DATA_BLOCK "DigiforceMain_DB"   // DB47
VERSION : 0.1
// stored: AutoNumber true, DBAccessibleFromOPCUA true, DBAccessibleFromWebserver true, InstanceOfName DigiforceMain, InstanceOfType FB
"DigiforceMain"
BEGIN
   Digiforce1_Instance.DataRead := 488;
   Digiforce1_Instance.DataWrite := 487;
   Digiforce1_Instance.send.Tare_X := FALSE;
   Digiforce1_Instance.send.Res_Stat := FALSE;
   Digiforce1_Instance.send.Stest := FALSE;
   Digiforce1_Instance.send.Strobe := FALSE;
   Digiforce1_Instance.send.Auto := FALSE;
   Digiforce1_Instance.send.reserve1 := FALSE;
   Digiforce1_Instance.send.reserve2 := FALSE;
   Digiforce1_Instance.send.reserve3 := FALSE;
   Digiforce1_Instance.send.Prog := 16#00;
   Digiforce1_Instance.send.Start := FALSE;
   Digiforce1_Instance.receive.dataD.Ready := TRUE;
   Digiforce1_Instance.receive.dataD.OK := FALSE;
   Digiforce1_Instance.receive.dataD.NOK := TRUE;
   Digiforce1_Instance.receive.dataD.NOK_ONL := FALSE;
   Digiforce1_Instance.receive.dataD.S1 := TRUE;
   Digiforce1_Instance.receive.dataD.S2 := FALSE;
   Digiforce1_Instance.receive.dataD.OK_STEST := FALSE;
   Digiforce1_Instance.receive.dataD.MEAS_ACT := FALSE;
   Digiforce1_Instance.receive.dataD.Strobe := FALSE;
   Digiforce1_Instance.receive.dataD.Prog0 := FALSE;
   Digiforce1_Instance.receive.dataD.Prog1 := FALSE;
   Digiforce1_Instance.receive.dataD.Prog2 := FALSE;
   Digiforce1_Instance.receive.dataD.reserve1 := FALSE;
   Digiforce1_Instance.receive.dataD.reserve2 := FALSE;
   Digiforce1_Instance.receive.dataD.reserve3 := FALSE;
   Digiforce1_Instance.receive.dataD.reserve4 := FALSE;
   Digiforce1_Instance.receive.dataD.Global_NOK := TRUE;
   Digiforce1_Instance.receive.dataD."Overload _NOK" := FALSE;
   Digiforce1_Instance.receive.dataD.Window_1_NOK := TRUE;
   Digiforce1_Instance.receive.dataD.Window_2_NOK := FALSE;
   Digiforce1_Instance.receive.dataD.Window_3_NOK := FALSE;
   Digiforce1_Instance.receive.dataD.Threshold_1_NOK := TRUE;
   Digiforce1_Instance.receive.dataD.Threshold_2_NOK := FALSE;
   Digiforce1_Instance.receive.dataD.Trapezoid_1_NOK := FALSE;
   Digiforce1_Instance.receive.dataD.Trapezoid2_NOK := FALSE;
   Digiforce1_Instance.receive.dataD.Envelope_NOK := FALSE;
   Digiforce1_Instance.receive.dataD."Measurement_w/o_READY" := FALSE;
   Digiforce1_Instance.receive.dataD.USB_logging_error := FALSE;
   Digiforce1_Instance.receive.dataD.reserve5 := FALSE;
   Digiforce1_Instance.receive.dataD.reserve6 := FALSE;
   Digiforce1_Instance.receive.dataD.reserve7 := FALSE;
   Digiforce1_Instance.receive.dataD.reserve8 := FALSE;
   Digiforce1_Instance.receive.dataA[1..20] := 909090.0;
   Digiforce1_Instance.receive.dataA[21] := 8.063384;
   Digiforce1_Instance.receive.dataA[22] := -0.03242895;
   Digiforce1_Instance.IEC_Timer_zmenaProgramu.PT := T#0MS;
   Digiforce1_Instance.IEC_Timer_zmenaProgramu.IN := FALSE;
   Digiforce2_Instance.DataRead := 548;
   Digiforce2_Instance.DataWrite := 547;
   Digiforce2_Instance.send.Tare_X := FALSE;
   Digiforce2_Instance.send.Res_Stat := FALSE;
   Digiforce2_Instance.send.Stest := FALSE;
   Digiforce2_Instance.send.Strobe := FALSE;
   Digiforce2_Instance.send.Auto := FALSE;
   Digiforce2_Instance.send.reserve1 := FALSE;
   Digiforce2_Instance.send.reserve2 := FALSE;
   Digiforce2_Instance.send.reserve3 := FALSE;
   Digiforce2_Instance.send.Prog := 16#00;
   Digiforce2_Instance.send.Start := FALSE;
   Digiforce2_Instance.receive.dataD.Ready := TRUE;
   Digiforce2_Instance.receive.dataD.OK := FALSE;
   Digiforce2_Instance.receive.dataD.NOK := TRUE;
   Digiforce2_Instance.receive.dataD.NOK_ONL := FALSE;
   Digiforce2_Instance.receive.dataD.S1 := TRUE;
   Digiforce2_Instance.receive.dataD.S2 := FALSE;
   Digiforce2_Instance.receive.dataD.OK_STEST := FALSE;
   Digiforce2_Instance.receive.dataD.MEAS_ACT := FALSE;
   Digiforce2_Instance.receive.dataD.Strobe := FALSE;
   Digiforce2_Instance.receive.dataD.Prog0 := FALSE;
   Digiforce2_Instance.receive.dataD.Prog1 := FALSE;
   Digiforce2_Instance.receive.dataD.Prog2 := FALSE;
   Digiforce2_Instance.receive.dataD.reserve1 := FALSE;
   Digiforce2_Instance.receive.dataD.reserve2 := FALSE;
   Digiforce2_Instance.receive.dataD.reserve3 := FALSE;
   Digiforce2_Instance.receive.dataD.reserve4 := FALSE;
   Digiforce2_Instance.receive.dataD.Global_NOK := TRUE;
   Digiforce2_Instance.receive.dataD."Overload _NOK" := FALSE;
   Digiforce2_Instance.receive.dataD.Window_1_NOK := TRUE;
   Digiforce2_Instance.receive.dataD.Window_2_NOK := FALSE;
   Digiforce2_Instance.receive.dataD.Window_3_NOK := FALSE;
   Digiforce2_Instance.receive.dataD.Threshold_1_NOK := TRUE;
   Digiforce2_Instance.receive.dataD.Threshold_2_NOK := FALSE;
   Digiforce2_Instance.receive.dataD.Trapezoid_1_NOK := FALSE;
   Digiforce2_Instance.receive.dataD.Trapezoid2_NOK := FALSE;
   Digiforce2_Instance.receive.dataD.Envelope_NOK := FALSE;
   Digiforce2_Instance.receive.dataD."Measurement_w/o_READY" := FALSE;
   Digiforce2_Instance.receive.dataD.USB_logging_error := FALSE;
   Digiforce2_Instance.receive.dataD.reserve5 := FALSE;
   Digiforce2_Instance.receive.dataD.reserve6 := FALSE;
   Digiforce2_Instance.receive.dataD.reserve7 := FALSE;
   Digiforce2_Instance.receive.dataD.reserve8 := FALSE;
   Digiforce2_Instance.receive.dataA[1..20] := 909090.0;
   Digiforce2_Instance.receive.dataA[21] := 8.028815;
   Digiforce2_Instance.receive.dataA[22] := -0.02130306;
   Digiforce2_Instance.IEC_Timer_zmenaProgramu.PT := T#0MS;
   Digiforce2_Instance.IEC_Timer_zmenaProgramu.IN := FALSE;
   Digiforce3_Instance.DataRead := 610;
   Digiforce3_Instance.DataWrite := 609;
   Digiforce3_Instance.send.Tare_X := FALSE;
   Digiforce3_Instance.send.Res_Stat := FALSE;
   Digiforce3_Instance.send.Stest := FALSE;
   Digiforce3_Instance.send.Strobe := FALSE;
   Digiforce3_Instance.send.Auto := FALSE;
   Digiforce3_Instance.send.reserve1 := FALSE;
   Digiforce3_Instance.send.reserve2 := FALSE;
   Digiforce3_Instance.send.reserve3 := FALSE;
   Digiforce3_Instance.send.Prog := 16#01;
   Digiforce3_Instance.send.Start := FALSE;
   Digiforce3_Instance.receive.dataD.Ready := TRUE;
   Digiforce3_Instance.receive.dataD.OK := FALSE;
   Digiforce3_Instance.receive.dataD.NOK := TRUE;
   Digiforce3_Instance.receive.dataD.NOK_ONL := FALSE;
   Digiforce3_Instance.receive.dataD.S1 := TRUE;
   Digiforce3_Instance.receive.dataD.S2 := FALSE;
   Digiforce3_Instance.receive.dataD.OK_STEST := FALSE;
   Digiforce3_Instance.receive.dataD.MEAS_ACT := FALSE;
   Digiforce3_Instance.receive.dataD.Strobe := FALSE;
   Digiforce3_Instance.receive.dataD.Prog0 := TRUE;
   Digiforce3_Instance.receive.dataD.Prog1 := FALSE;
   Digiforce3_Instance.receive.dataD.Prog2 := FALSE;
   Digiforce3_Instance.receive.dataD.reserve1 := FALSE;
   Digiforce3_Instance.receive.dataD.reserve2 := FALSE;
   Digiforce3_Instance.receive.dataD.reserve3 := FALSE;
   Digiforce3_Instance.receive.dataD.reserve4 := FALSE;
   Digiforce3_Instance.receive.dataD.Global_NOK := TRUE;
   Digiforce3_Instance.receive.dataD."Overload _NOK" := FALSE;
   Digiforce3_Instance.receive.dataD.Window_1_NOK := TRUE;
   Digiforce3_Instance.receive.dataD.Window_2_NOK := FALSE;
   Digiforce3_Instance.receive.dataD.Window_3_NOK := FALSE;
   Digiforce3_Instance.receive.dataD.Threshold_1_NOK := TRUE;
   Digiforce3_Instance.receive.dataD.Threshold_2_NOK := FALSE;
   Digiforce3_Instance.receive.dataD.Trapezoid_1_NOK := FALSE;
   Digiforce3_Instance.receive.dataD.Trapezoid2_NOK := FALSE;
   Digiforce3_Instance.receive.dataD.Envelope_NOK := FALSE;
   Digiforce3_Instance.receive.dataD."Measurement_w/o_READY" := FALSE;
   Digiforce3_Instance.receive.dataD.USB_logging_error := FALSE;
   Digiforce3_Instance.receive.dataD.reserve5 := FALSE;
   Digiforce3_Instance.receive.dataD.reserve6 := FALSE;
   Digiforce3_Instance.receive.dataD.reserve7 := FALSE;
   Digiforce3_Instance.receive.dataD.reserve8 := FALSE;
   Digiforce3_Instance.receive.dataA[1..20] := 909090.0;
   Digiforce3_Instance.receive.dataA[21] := 8.030701;
   Digiforce3_Instance.receive.dataA[22] := -0.01457718;
   Digiforce3_Instance.IEC_Timer_zmenaProgramu.PT := T#10S;
   Digiforce3_Instance.IEC_Timer_zmenaProgramu.IN := FALSE;
   Digiforce4_Instance.DataRead := 672;
   Digiforce4_Instance.DataWrite := 671;
   Digiforce4_Instance.send.Tare_X := FALSE;
   Digiforce4_Instance.send.Res_Stat := FALSE;
   Digiforce4_Instance.send.Stest := FALSE;
   Digiforce4_Instance.send.Strobe := FALSE;
   Digiforce4_Instance.send.Auto := FALSE;
   Digiforce4_Instance.send.reserve1 := FALSE;
   Digiforce4_Instance.send.reserve2 := FALSE;
   Digiforce4_Instance.send.reserve3 := FALSE;
   Digiforce4_Instance.send.Prog := 16#01;
   Digiforce4_Instance.send.Start := FALSE;
   Digiforce4_Instance.receive.dataD.Ready := TRUE;
   Digiforce4_Instance.receive.dataD.OK := FALSE;
   Digiforce4_Instance.receive.dataD.NOK := TRUE;
   Digiforce4_Instance.receive.dataD.NOK_ONL := FALSE;
   Digiforce4_Instance.receive.dataD.S1 := TRUE;
   Digiforce4_Instance.receive.dataD.S2 := FALSE;
   Digiforce4_Instance.receive.dataD.OK_STEST := FALSE;
   Digiforce4_Instance.receive.dataD.MEAS_ACT := FALSE;
   Digiforce4_Instance.receive.dataD.Strobe := FALSE;
   Digiforce4_Instance.receive.dataD.Prog0 := TRUE;
   Digiforce4_Instance.receive.dataD.Prog1 := FALSE;
   Digiforce4_Instance.receive.dataD.Prog2 := FALSE;
   Digiforce4_Instance.receive.dataD.reserve1 := FALSE;
   Digiforce4_Instance.receive.dataD.reserve2 := FALSE;
   Digiforce4_Instance.receive.dataD.reserve3 := FALSE;
   Digiforce4_Instance.receive.dataD.reserve4 := FALSE;
   Digiforce4_Instance.receive.dataD.Global_NOK := TRUE;
   Digiforce4_Instance.receive.dataD."Overload _NOK" := FALSE;
   Digiforce4_Instance.receive.dataD.Window_1_NOK := TRUE;
   Digiforce4_Instance.receive.dataD.Window_2_NOK := FALSE;
   Digiforce4_Instance.receive.dataD.Window_3_NOK := FALSE;
   Digiforce4_Instance.receive.dataD.Threshold_1_NOK := TRUE;
   Digiforce4_Instance.receive.dataD.Threshold_2_NOK := FALSE;
   Digiforce4_Instance.receive.dataD.Trapezoid_1_NOK := FALSE;
   Digiforce4_Instance.receive.dataD.Trapezoid2_NOK := FALSE;
   Digiforce4_Instance.receive.dataD.Envelope_NOK := FALSE;
   Digiforce4_Instance.receive.dataD."Measurement_w/o_READY" := FALSE;
   Digiforce4_Instance.receive.dataD.USB_logging_error := FALSE;
   Digiforce4_Instance.receive.dataD.reserve5 := FALSE;
   Digiforce4_Instance.receive.dataD.reserve6 := FALSE;
   Digiforce4_Instance.receive.dataD.reserve7 := FALSE;
   Digiforce4_Instance.receive.dataD.reserve8 := FALSE;
   Digiforce4_Instance.receive.dataA[1..20] := 909090.0;
   Digiforce4_Instance.receive.dataA[21] := 8.018154;
   Digiforce4_Instance.receive.dataA[22] := -0.01945436;
   Digiforce4_Instance.IEC_Timer_zmenaProgramu.PT := T#10S;
   Digiforce4_Instance.IEC_Timer_zmenaProgramu.IN := FALSE;
END_DATA_BLOCK

DATA_BLOCK "RivetingHistoryLeft_DB"   // DB41
VERSION : 0.1
// stored: AutoNumber true, DBAccessibleFromOPCUA true, DBAccessibleFromWebserver true, InstanceOfName RivetingHistory, InstanceOfType FB
"RivetingHistory"
BEGIN
   history[0..99].Start := FALSE;
   history[0..24].PrgNumber := 2;
   history[25..99].PrgNumber := 0;
   history[0..14].Ready := TRUE;
   history[15].Ready := FALSE;
   history[16..24].Ready := TRUE;
   history[25..99].Ready := FALSE;
   history[0..99].Running := FALSE;
   history[0..4].OK := TRUE;
   history[5..9].OK := FALSE;
   history[10..11].OK := TRUE;
   history[12..13].OK := FALSE;
   history[14..24].OK := TRUE;
   history[25..99].OK := FALSE;
   history[0..4].NOK := FALSE;
   history[5..9].NOK := TRUE;
   history[10..11].NOK := FALSE;
   history[12..13].NOK := TRUE;
   history[14..99].NOK := FALSE;
   history[0..24].H1OK := TRUE;
   history[25..99].H1OK := FALSE;
   history[0..4].H2OK := TRUE;
   history[5..9].H2OK := FALSE;
   history[10..11].H2OK := TRUE;
   history[12..13].H2OK := FALSE;
   history[14..24].H2OK := TRUE;
   history[25..99].H2OK := FALSE;
   history[0..4].TimeOK := TRUE;
   history[5..9].TimeOK := FALSE;
   history[10..11].TimeOK := TRUE;
   history[12..13].TimeOK := FALSE;
   history[14..24].TimeOK := TRUE;
   history[25..99].TimeOK := FALSE;
   history[0..99].StartError := FALSE;
   history[0..99].LastH1 := 0.0;
   history[0..3].LastH2 := 0.0;
   history[4].LastH2 := 2.23;
   history[5..9].LastH2 := 0.0;
   history[10].LastH2 := 2.29;
   history[11].LastH2 := 2.22;
   history[12..13].LastH2 := 0.0;
   history[14].LastH2 := 2.27;
   history[15..16].LastH2 := 2.25;
   history[17].LastH2 := 2.4;
   history[18].LastH2 := 2.28;
   history[19].LastH2 := 2.39;
   history[20].LastH2 := 2.4;
   history[21].LastH2 := 2.39;
   history[22].LastH2 := 2.37;
   history[23..24].LastH2 := 2.4;
   history[25..99].LastH2 := 0.0;
   history[0..18].LastTime := 0.0;
   history[19..21].LastTime := 0.12;
   history[22..23].LastTime := 0.0;
   history[24].LastTime := 0.12;
   history[25..99].LastTime := 0.0;
   history[0].LastZ1 := 11.69;
   history[1].LastZ1 := 11.86;
   history[2].LastZ1 := 11.77;
   history[3].LastZ1 := 11.85;
   history[4].LastZ1 := 12.06;
   history[5].LastZ1 := 11.86;
   history[6].LastZ1 := 11.68;
   history[7].LastZ1 := 11.85;
   history[8].LastZ1 := 11.74;
   history[9].LastZ1 := 11.89;
   history[10].LastZ1 := 12.16;
   history[11].LastZ1 := 12.09;
   history[12].LastZ1 := 11.76;
   history[13].LastZ1 := 11.73;
   history[14].LastZ1 := 12.09;
   history[15..16].LastZ1 := 12.38;
   history[17].LastZ1 := 12.19;
   history[18].LastZ1 := 12.4;
   history[19..24].LastZ1 := 12.2;
   history[25..99].LastZ1 := 0.0;
   history[0..99].Error := FALSE;
   history[0..99].NewData := FALSE;
   history[0..4].Z1OK := TRUE;
   history[5..9].Z1OK := FALSE;
   history[10..11].Z1OK := TRUE;
   history[12..13].Z1OK := FALSE;
   history[14..24].Z1OK := TRUE;
   history[25..99].Z1OK := FALSE;
   history[0..24].NewDataAfterStart := TRUE;
   history[25..99].NewDataAfterStart := FALSE;
   history[0].LastZ2 := 11.69;
   history[1].LastZ2 := 11.86;
   history[2].LastZ2 := 11.77;
   history[3].LastZ2 := 11.85;
   history[4..99].LastZ2 := 0.0;
END_DATA_BLOCK

DATA_BLOCK "RivetingHistoryRight_DB"   // DB23
VERSION : 0.1
// stored: AutoNumber true, DBAccessibleFromOPCUA true, DBAccessibleFromWebserver true, InstanceOfName RivetingHistory, InstanceOfType FB
"RivetingHistory"
BEGIN
   history[0..99].Start := FALSE;
   history[0..24].PrgNumber := 2;
   history[25..52].PrgNumber := 1;
   history[53..66].PrgNumber := 2;
   history[67].PrgNumber := 1;
   history[68..99].PrgNumber := 0;
   history[0..11].Ready := TRUE;
   history[12].Ready := FALSE;
   history[13..67].Ready := TRUE;
   history[68..99].Ready := FALSE;
   history[0..99].Running := FALSE;
   history[0..19].OK := TRUE;
   history[20..22].OK := FALSE;
   history[23].OK := TRUE;
   history[24].OK := FALSE;
   history[25..32].OK := TRUE;
   history[33].OK := FALSE;
   history[34..35].OK := TRUE;
   history[36].OK := FALSE;
   history[37..43].OK := TRUE;
   history[44..99].OK := FALSE;
   history[0..19].NOK := FALSE;
   history[20..22].NOK := TRUE;
   history[23].NOK := FALSE;
   history[24].NOK := TRUE;
   history[25..32].NOK := FALSE;
   history[33].NOK := TRUE;
   history[34..35].NOK := FALSE;
   history[36].NOK := TRUE;
   history[37..43].NOK := FALSE;
   history[44..67].NOK := TRUE;
   history[68..99].NOK := FALSE;
   history[0..32].H1OK := TRUE;
   history[33].H1OK := FALSE;
   history[34..35].H1OK := TRUE;
   history[36].H1OK := FALSE;
   history[37..55].H1OK := TRUE;
   history[56..99].H1OK := FALSE;
   history[0..19].H2OK := TRUE;
   history[20..22].H2OK := FALSE;
   history[23].H2OK := TRUE;
   history[24].H2OK := FALSE;
   history[25..32].H2OK := TRUE;
   history[33].H2OK := FALSE;
   history[34..35].H2OK := TRUE;
   history[36].H2OK := FALSE;
   history[37..43].H2OK := TRUE;
   history[44..99].H2OK := FALSE;
   history[0..23].TimeOK := TRUE;
   history[24].TimeOK := FALSE;
   history[25..32].TimeOK := TRUE;
   history[33].TimeOK := FALSE;
   history[34..35].TimeOK := TRUE;
   history[36].TimeOK := FALSE;
   history[37..43].TimeOK := TRUE;
   history[44..99].TimeOK := FALSE;
   history[0..99].StartError := FALSE;
   history[0..24].LastH1 := 0.0;
   history[25].LastH1 := 5.09;
   history[26].LastH1 := 5.17;
   history[27].LastH1 := 5.11;
   history[28].LastH1 := 5.29;
   history[29].LastH1 := 5.23;
   history[30].LastH1 := 5.18;
   history[31].LastH1 := 5.22;
   history[32].LastH1 := 5.0;
   history[33].LastH1 := 4.84;
   history[34].LastH1 := 5.27;
   history[35].LastH1 := 5.26;
   history[36].LastH1 := -0.11;
   history[37].LastH1 := 5.25;
   history[38].LastH1 := 2.47;
   history[39..99].LastH1 := 0.0;
   history[0..3].LastH2 := 0.0;
   history[4].LastH2 := 2.37;
   history[5..6].LastH2 := 2.38;
   history[7..8].LastH2 := 2.4;
   history[9].LastH2 := 2.39;
   history[10].LastH2 := 2.38;
   history[11].LastH2 := 2.4;
   history[12..13].LastH2 := 2.39;
   history[14].LastH2 := 0.19;
   history[15].LastH2 := 2.39;
   history[16..17].LastH2 := 0.19;
   history[18].LastH2 := 0.18;
   history[19].LastH2 := 0.19;
   history[20].LastH2 := 0.18;
   history[21].LastH2 := 0.19;
   history[22].LastH2 := 0.18;
   history[23].LastH2 := 2.37;
   history[24].LastH2 := 0.0;
   history[25..26].LastH2 := 2.38;
   history[27].LastH2 := 2.36;
   history[28].LastH2 := 2.4;
   history[29].LastH2 := 2.39;
   history[30].LastH2 := 2.38;
   history[31].LastH2 := 2.33;
   history[32].LastH2 := 2.38;
   history[33].LastH2 := 0.0;
   history[34].LastH2 := 2.4;
   history[35].LastH2 := 2.39;
   history[36].LastH2 := 0.0;
   history[37].LastH2 := 2.39;
   history[38].LastH2 := 2.4;
   history[39].LastH2 := 2.39;
   history[40].LastH2 := 2.4;
   history[41].LastH2 := 2.38;
   history[42].LastH2 := 2.39;
   history[43].LastH2 := 2.4;
   history[44..99].LastH2 := 0.0;
   history[0..3].LastTime := 0.0;
   history[4].LastTime := 1.47;
   history[5].LastTime := 0.96;
   history[6].LastTime := 0.98;
   history[7].LastTime := 0.65;
   history[8].LastTime := 0.68;
   history[9].LastTime := 1.01;
   history[10].LastTime := 0.94;
   history[11].LastTime := 0.86;
   history[12..13].LastTime := 0.15;
   history[14].LastTime := 0.0;
   history[15].LastTime := 0.33;
   history[16..22].LastTime := 0.0;
   history[23].LastTime := 0.83;
   history[24].LastTime := 0.0;
   history[25].LastTime := 1.94;
   history[26].LastTime := 2.55;
   history[27].LastTime := 2.14;
   history[28].LastTime := 2.35;
   history[29].LastTime := 2.7;
   history[30].LastTime := 2.31;
   history[31].LastTime := 2.17;
   history[32].LastTime := 2.47;
   history[33].LastTime := 0.0;
   history[34].LastTime := 2.34;
   history[35].LastTime := 2.88;
   history[36].LastTime := 0.0;
   history[37].LastTime := 2.21;
   history[38].LastTime := 0.12;
   history[39].LastTime := 2.58;
   history[40].LastTime := 2.51;
   history[41].LastTime := 2.3;
   history[42].LastTime := 2.34;
   history[43].LastTime := 2.54;
   history[44..99].LastTime := 0.0;
   history[0].LastZ1 := 11.96;
   history[1].LastZ1 := 12.01;
   history[2].LastZ1 := 12.11;
   history[3].LastZ1 := 12.1;
   history[4].LastZ1 := 12.38;
   history[5..6].LastZ1 := 12.2;
   history[7].LastZ1 := 12.14;
   history[8].LastZ1 := 12.13;
   history[9].LastZ1 := 12.19;
   history[10].LastZ1 := 12.0;
   history[11].LastZ1 := 12.18;
   history[12..13].LastZ1 := 12.58;
   history[14].LastZ1 := 12.33;
   history[15].LastZ1 := 12.6;
   history[16].LastZ1 := 12.34;
   history[17].LastZ1 := 12.33;
   history[18].LastZ1 := 12.32;
   history[19..20].LastZ1 := 12.3;
   history[21].LastZ1 := 12.33;
   history[22].LastZ1 := 12.3;
   history[23..24].LastZ1 := 12.43;
   history[25].LastZ1 := 15.42;
   history[26].LastZ1 := 15.4;
   history[27].LastZ1 := 15.41;
   history[28].LastZ1 := 15.4;
   history[29].LastZ1 := 15.39;
   history[30].LastZ1 := 15.4;
   history[31].LastZ1 := 15.39;
   history[32].LastZ1 := 15.42;
   history[33].LastZ1 := 15.43;
   history[34].LastZ1 := 15.41;
   history[35].LastZ1 := 15.44;
   history[36].LastZ1 := 8.43;
   history[37].LastZ1 := 15.42;
   history[38].LastZ1 := 12.39;
   history[39].LastZ1 := 15.39;
   history[40].LastZ1 := 15.46;
   history[41].LastZ1 := 15.42;
   history[42].LastZ1 := 15.43;
   history[43].LastZ1 := 15.39;
   history[44].LastZ1 := 13.18;
   history[45..47].LastZ1 := 13.2;
   history[48].LastZ1 := 3.22;
   history[49..99].LastZ1 := 0.0;
   history[0..99].Error := FALSE;
   history[0..99].NewData := FALSE;
   history[0..23].Z1OK := TRUE;
   history[24].Z1OK := FALSE;
   history[25..35].Z1OK := TRUE;
   history[36].Z1OK := FALSE;
   history[37..43].Z1OK := TRUE;
   history[44..99].Z1OK := FALSE;
   history[0..48].NewDataAfterStart := TRUE;
   history[49..99].NewDataAfterStart := FALSE;
   history[0].LastZ2 := 11.96;
   history[1].LastZ2 := 12.01;
   history[2].LastZ2 := 12.11;
   history[3].LastZ2 := 12.1;
   history[4..99].LastZ2 := 0.0;
END_DATA_BLOCK

DATA_BLOCK "FittingHistoryLeftCupforming_DB"   // DB35
VERSION : 0.1
// stored: AutoNumber true, DBAccessibleFromOPCUA true, DBAccessibleFromWebserver true, InstanceOfName FittingHistory, InstanceOfType FB
"FittingHistory"
   // VAR_INPUT
   //    iNewCycle : Bool;
   //    iData : "UDT_Results_Cupforming";
   // END_VAR
   // VAR RETAIN
   //    history : Array[0..99] of "UDT_Results_Cupforming";
   // END_VAR
   // VAR
   //    pageData { S7_SetPoint := 'True'} : Array[0..9] of "UDT_Results_Cupforming";
   // END_VAR
   // VAR RETAIN
   //    pageNumber { S7_SetPoint := 'True'} : USInt := 0;
   // END_VAR
   // VAR
   //    resetHistory : Bool;
   //    R_TRIG_Instance { S7_SetPoint := 'True'} : R_TRIG;
   // END_VAR
BEGIN
   history[0].MaxForce := -7.98946;
   history[1].MaxForce := -7.998657;
   history[2].MaxForce := -7.98946;
   history[3..4].MaxForce := -7.984862;
   history[5].MaxForce := -8.007853;
   history[6].MaxForce := -7.994059;
   history[7].MaxForce := -7.980264;
   history[8].MaxForce := 32.33566;
   history[9].MaxForce := 30.64817;
   history[10].MaxForce := 27.33296;
   history[11..99].MaxForce := 0.0;
   history[0].MinimalWay := 9.841429;
   history[1].MinimalWay := 9.875875;
   history[2].MinimalWay := 9.837013;
   history[3].MinimalWay := 9.846728;
   history[4].MinimalWay := 9.887358;
   history[5].MinimalWay := 9.779602;
   history[6].MinimalWay := 9.831714;
   history[7].MinimalWay := 9.859094;
   history[8].MinimalWay := 8.49007;
   history[9].MinimalWay := 8.491837;
   history[10].MinimalWay := 8.488304;
   history[11..99].MinimalWay := 0.0;
   history[0].MaxZposition := 55.44488;
   history[1].MaxZposition := 55.55556;
   history[2].MaxZposition := 55.54471;
   history[3].MaxZposition := 55.3928;
   history[4].MaxZposition := 55.42969;
   history[5].MaxZposition := 55.67492;
   history[6].MaxZposition := 55.59462;
   history[7].MaxZposition := 55.36676;
   history[8].MaxZposition := 59.20356;
   history[9].MaxZposition := 59.29688;
   history[10].MaxZposition := 59.16667;
   history[11..99].MaxZposition := 0.0;
   history[0..10].OK := TRUE;
   history[11..99].OK := FALSE;
   history[0..99].NOK := FALSE;
   history[0..10].parameters.DigiforceProgram := 1;
   history[11..99].parameters.DigiforceProgram := 0;
   history[0..10].parameters.FinalSpeed := 20.0;
   history[11..99].parameters.FinalSpeed := 0.0;
   history[0..10].parameters.ApproachSpeed := 100.0;
   history[11..99].parameters.ApproachSpeed := 0.0;
   history[0..7].parameters.FinalForce := 80.0;
   history[8..10].parameters.FinalForce := 90.0;
   history[11..99].parameters.FinalForce := 0.0;
   history[0..10].parameters.ApproachForce := 20.0;
   history[11..99].parameters.ApproachForce := 0.0;
   history[0..7].parameters.EndWayImmediate := 9.9;
   history[8..10].parameters.EndWayImmediate := 8.5;
   history[11..99].parameters.EndWayImmediate := 0.0;
   history[0..7].parameters.EndWayWithTimeout := 9.9;
   history[8..9].parameters.EndWayWithTimeout := 8.6;
   history[10].parameters.EndWayWithTimeout := 8.5;
   history[11..99].parameters.EndWayWithTimeout := 0.0;
   history[0..7].parameters.SwitchingWay := 50.0;
   history[8..10].parameters.SwitchingWay := 53.0;
   history[11..99].parameters.SwitchingWay := 0.0;
   history[0..10].parameters.EndWayTimeout := T#300MS;
   history[11..99].parameters.EndWayTimeout := T#0MS;
END_DATA_BLOCK

DATA_BLOCK "FittingHistoryRightCupforming_DB"   // DB43
VERSION : 0.1
// stored: AutoNumber true, DBAccessibleFromOPCUA true, DBAccessibleFromWebserver true, InstanceOfName FittingHistory, InstanceOfType FB
"FittingHistory"
   // VAR_INPUT
   //    iNewCycle : Bool;
   //    iData : "UDT_Results_Cupforming";
   // END_VAR
   // VAR RETAIN
   //    history : Array[0..99] of "UDT_Results_Cupforming";
   // END_VAR
   // VAR
   //    pageData { S7_SetPoint := 'True'} : Array[0..9] of "UDT_Results_Cupforming";
   // END_VAR
   // VAR RETAIN
   //    pageNumber { S7_SetPoint := 'True'} : USInt := 0;
   // END_VAR
   // VAR
   //    resetHistory : Bool;
   //    R_TRIG_Instance { S7_SetPoint := 'True'} : R_TRIG;
   // END_VAR
BEGIN
   history[0].MaxForce := 8.163286;
   history[1].MaxForce := 8.130146;
   history[2..3].MaxForce := 8.158552;
   history[4..5].MaxForce := 8.177489;
   history[6].MaxForce := 8.149084;
   history[7].MaxForce := 8.158552;
   history[8].MaxForce := 54.72517;
   history[9].MaxForce := 54.91927;
   history[10].MaxForce := 52.27753;
   history[11..99].MaxForce := 0.0;
   history[0].MinimalWay := 9.87697;
   history[1].MinimalWay := 9.87257;
   history[2].MinimalWay := 9.886649;
   history[3].MinimalWay := 9.885769;
   history[4].MinimalWay := 9.896328;
   history[5].MinimalWay := 9.890168;
   history[6].MinimalWay := 9.88137;
   history[7].MinimalWay := 9.887528;
   history[8].MinimalWay := 9.091208;
   history[9].MinimalWay := 8.947783;
   history[10].MinimalWay := 8.997938;
   history[11..99].MinimalWay := 0.0;
   history[0].MaxZposition := 56.52127;
   history[1].MaxZposition := 56.64497;
   history[2].MaxZposition := 56.6059;
   history[3].MaxZposition := 56.54731;
   history[4].MaxZposition := 56.57769;
   history[5].MaxZposition := 56.63412;
   history[6].MaxZposition := 56.4974;
   history[7].MaxZposition := 56.69054;
   history[8].MaxZposition := 58.5612;
   history[9].MaxZposition := 58.33334;
   history[10].MaxZposition := 58.6849;
   history[11..99].MaxZposition := 0.0;
   history[0..10].OK := TRUE;
   history[11..99].OK := FALSE;
   history[0..99].NOK := FALSE;
   history[0..10].parameters.DigiforceProgram := 1;
   history[11..99].parameters.DigiforceProgram := 0;
   history[0..10].parameters.FinalSpeed := 20.0;
   history[11..99].parameters.FinalSpeed := 0.0;
   history[0..10].parameters.ApproachSpeed := 100.0;
   history[11..99].parameters.ApproachSpeed := 0.0;
   history[0..7].parameters.FinalForce := 80.0;
   history[8..10].parameters.FinalForce := 90.0;
   history[11..99].parameters.FinalForce := 0.0;
   history[0..10].parameters.ApproachForce := 20.0;
   history[11..99].parameters.ApproachForce := 0.0;
   history[0..7].parameters.EndWayImmediate := 9.9;
   history[8..10].parameters.EndWayImmediate := 9.0;
   history[11..99].parameters.EndWayImmediate := 0.0;
   history[0..7].parameters.EndWayWithTimeout := 9.9;
   history[8..9].parameters.EndWayWithTimeout := 9.1;
   history[10].parameters.EndWayWithTimeout := 9.0;
   history[11..99].parameters.EndWayWithTimeout := 0.0;
   history[0..7].parameters.SwitchingWay := 50.0;
   history[8..10].parameters.SwitchingWay := 53.0;
   history[11..99].parameters.SwitchingWay := 0.0;
   history[0..10].parameters.EndWayTimeout := T#300MS;
   history[11..99].parameters.EndWayTimeout := T#0MS;
END_DATA_BLOCK

DATA_BLOCK "HydraulicMain_DB"   // DB55
VERSION : 0.1
// stored: AutoNumber true, DBAccessibleFromOPCUA true, DBAccessibleFromWebserver true, InstanceOfName HydraulicMain, InstanceOfType FB
"HydraulicMain"
   // VAR
   //    HydraulicCylinder_LeftCupforming { S7_SetPoint := 'True'} : "HydraulicCylinder";
   //    HydraulicCylinder_RightCupforming { S7_SetPoint := 'True'} : "HydraulicCylinder";
   //    VH1StatusOld { S7_SetPoint := 'True'} : "UDT_Cylinder";
   //    VH2StatusOld { S7_SetPoint := 'True'} : "UDT_Cylinder";
   //    VH3StatusOld { S7_SetPoint := 'True'} : "UDT_Cylinder";
   //    VH4StatusOld { S7_SetPoint := 'True'} : "UDT_Cylinder";
   //    FittingCycle_InstanceCupformingLeft { S7_SetPoint := 'True'} : "FittingCycle";
   //    FittingCycle_InstanceCupformingRight { S7_SetPoint := 'True'} : "FittingCycle";
   //    R_TRIG_Instance { S7_SetPoint := 'True'} : R_TRIG;
   //    R_TRIG_Instance_1 { S7_SetPoint := 'True'} : R_TRIG;
   //    R_TRIG_Instance_2 { S7_SetPoint := 'True'} : R_TRIG;
   //    R_TRIG_Instance_3 { S7_SetPoint := 'True'} : R_TRIG;
   //    HydraulicMotor_Instance { S7_SetPoint := 'True'} : "HydraulicMotor";
   //    dummyCylinderLeft { ExternalAccessible := 'False'; ExternalVisible := 'False'; ExternalWritable := 'False'} : "UDT_Cylinder";
   //    dummyCylinderRight { S7_SetPoint := 'True'} : "UDT_Cylinder";
   // END_VAR
BEGIN
   HydraulicCylinder_LeftCupforming.HydraulicActive := FALSE;
   HydraulicCylinder_LeftCupforming.BasicPositionMin := -5.0;
   HydraulicCylinder_LeftCupforming.BasicPositionMax := 10.0;
   HydraulicCylinder_LeftCupforming.MaxPosition := 105.0;
   HydraulicCylinder_LeftCupforming.ManualCommand := 0;
   HydraulicCylinder_LeftCupforming.CylinderNumber := 3;
   HydraulicCylinder_LeftCupforming.dataOld.Pressure := 0.0;
   HydraulicCylinder_LeftCupforming.dataOld.Flow := 0.0;
   HydraulicCylinder_LeftCupforming.dataOld.Position := 0.0;
   HydraulicCylinder_LeftCupforming.dataOld.StandstillPosition := 0.0;
   HydraulicCylinder_LeftCupforming.dataOld.PressureCmd := 0.0;
   HydraulicCylinder_LeftCupforming.dataOld.FlowCmd := 0.0;
   HydraulicCylinder_LeftCupforming.dataOld.PressureBack := 0.0;
   HydraulicCylinder_LeftCupforming.dataOld.FlowBack := 0.0;
   HydraulicCylinder_LeftCupforming.dataOld.HAxis := 0.0;
   HydraulicCylinder_LeftCupforming.dataOld.Force := 0.0;
   HydraulicCylinder_LeftCupforming.dataOld.Status.InWp := FALSE;
   HydraulicCylinder_LeftCupforming.dataOld.Status.InBp := TRUE;
   HydraulicCylinder_LeftCupforming.dataOld.Status.InFp := TRUE;
   HydraulicCylinder_LeftCupforming.dataOld.Status.ToWp := FALSE;
   HydraulicCylinder_LeftCupforming.dataOld.Status.ToBp := FALSE;
   HydraulicCylinder_LeftCupforming.dataOld.Status.ToFp := TRUE;
   HydraulicCylinder_LeftCupforming.noCollision := TRUE;
   HydraulicCylinder_LeftCupforming.IEC_Timer_0_Instance.PT := T#3S;
   HydraulicCylinder_LeftCupforming.IEC_Timer_0_Instance.IN := FALSE;
   HydraulicCylinder_LeftCupforming.R_TRIG_Instance.CLK := TRUE;
   HydraulicCylinder_LeftCupforming.R_TRIG_Instance.Q := FALSE;
   HydraulicCylinder_LeftCupforming.R_TRIG_Instance.Stat_Bit := TRUE;
   HydraulicCylinder_LeftCupforming.difference := -0.01085043;
   HydraulicCylinder_LeftCupforming.re := -0.1085043;
   HydraulicCylinder_LeftCupforming.IEC_Timer_0_Instance_1.PT := T#400MS;
   HydraulicCylinder_LeftCupforming.IEC_Timer_0_Instance_1.IN := TRUE;
   HydraulicCylinder_LeftCupforming.RampFunction_Instance.Output := 0.0;
   HydraulicCylinder_LeftCupforming.RampFunction_Instance.ErrorBits := 16#0000_0000;
   HydraulicCylinder_RightCupforming.HydraulicActive := FALSE;
   HydraulicCylinder_RightCupforming.BasicPositionMin := -5.0;
   HydraulicCylinder_RightCupforming.BasicPositionMax := 10.0;
   HydraulicCylinder_RightCupforming.MaxPosition := 105.0;
   HydraulicCylinder_RightCupforming.ManualCommand := 0;
   HydraulicCylinder_RightCupforming.CylinderNumber := 4;
   HydraulicCylinder_RightCupforming.dataOld.Pressure := 0.0;
   HydraulicCylinder_RightCupforming.dataOld.Flow := 0.0;
   HydraulicCylinder_RightCupforming.dataOld.Position := 0.0;
   HydraulicCylinder_RightCupforming.dataOld.StandstillPosition := 0.0;
   HydraulicCylinder_RightCupforming.dataOld.PressureCmd := 0.0;
   HydraulicCylinder_RightCupforming.dataOld.FlowCmd := 0.0;
   HydraulicCylinder_RightCupforming.dataOld.PressureBack := 0.0;
   HydraulicCylinder_RightCupforming.dataOld.FlowBack := 0.0;
   HydraulicCylinder_RightCupforming.dataOld.HAxis := 0.0;
   HydraulicCylinder_RightCupforming.dataOld.Force := 0.0;
   HydraulicCylinder_RightCupforming.dataOld.Status.InWp := FALSE;
   HydraulicCylinder_RightCupforming.dataOld.Status.InBp := TRUE;
   HydraulicCylinder_RightCupforming.dataOld.Status.InFp := TRUE;
   HydraulicCylinder_RightCupforming.dataOld.Status.ToWp := FALSE;
   HydraulicCylinder_RightCupforming.dataOld.Status.ToBp := FALSE;
   HydraulicCylinder_RightCupforming.dataOld.Status.ToFp := TRUE;
   HydraulicCylinder_RightCupforming.noCollision := TRUE;
   HydraulicCylinder_RightCupforming.IEC_Timer_0_Instance.PT := T#3S;
   HydraulicCylinder_RightCupforming.IEC_Timer_0_Instance.IN := FALSE;
   HydraulicCylinder_RightCupforming.R_TRIG_Instance.CLK := TRUE;
   HydraulicCylinder_RightCupforming.R_TRIG_Instance.Q := FALSE;
   HydraulicCylinder_RightCupforming.R_TRIG_Instance.Stat_Bit := TRUE;
   HydraulicCylinder_RightCupforming.difference := -0.006510258;
   HydraulicCylinder_RightCupforming.re := -0.06510258;
   HydraulicCylinder_RightCupforming.IEC_Timer_0_Instance_1.PT := T#400MS;
   HydraulicCylinder_RightCupforming.IEC_Timer_0_Instance_1.IN := TRUE;
   HydraulicCylinder_RightCupforming.RampFunction_Instance.Output := 0.0;
   HydraulicCylinder_RightCupforming.RampFunction_Instance.ErrorBits := 16#0000_0000;
   VH1StatusOld.InWp := FALSE;
   VH1StatusOld.InBp := FALSE;
   VH1StatusOld.InFp := FALSE;
   VH1StatusOld.ToWp := FALSE;
   VH1StatusOld.ToBp := FALSE;
   VH1StatusOld.ToFp := FALSE;
   VH2StatusOld.InWp := FALSE;
   VH2StatusOld.InBp := FALSE;
   VH2StatusOld.InFp := FALSE;
   VH2StatusOld.ToWp := FALSE;
   VH2StatusOld.ToBp := FALSE;
   VH2StatusOld.ToFp := FALSE;
   VH3StatusOld.InWp := FALSE;
   VH3StatusOld.InBp := FALSE;
   VH3StatusOld.InFp := FALSE;
   VH3StatusOld.ToWp := FALSE;
   VH3StatusOld.ToBp := FALSE;
   VH3StatusOld.ToFp := FALSE;
   VH4StatusOld.InWp := FALSE;
   VH4StatusOld.InBp := FALSE;
   VH4StatusOld.InFp := FALSE;
   VH4StatusOld.ToWp := FALSE;
   VH4StatusOld.ToBp := FALSE;
   VH4StatusOld.ToFp := FALSE;
   FittingCycle_InstanceCupformingLeft.parameters.DigiforceProgram := 1;
   FittingCycle_InstanceCupformingLeft.parameters.FinalSpeed := 25.0;
   FittingCycle_InstanceCupformingLeft.parameters.ApproachSpeed := 25.0;
   FittingCycle_InstanceCupformingLeft.parameters.FinalForce := 10.0;
   FittingCycle_InstanceCupformingLeft.parameters.ApproachForce := 10.0;
   FittingCycle_InstanceCupformingLeft.parameters.EndWayImmediate := 2.55;
   FittingCycle_InstanceCupformingLeft.parameters.EndWayWithTimeout := 3.0;
   FittingCycle_InstanceCupformingLeft.parameters.SwitchingWay := 20.0;
   FittingCycle_InstanceCupformingLeft.parameters.EndWayTimeout := T#300MS;
   FittingCycle_InstanceCupformingLeft.basicPosition := TRUE;
   FittingCycle_InstanceCupformingLeft.MaxPosition := 105.0;
   FittingCycle_InstanceCupformingLeft.endStopCylinderActive := TRUE;
   FittingCycle_InstanceCupformingLeft.shiftSupportToWork := FALSE;
   FittingCycle_InstanceCupformingLeft.cnt := 0;
   FittingCycle_InstanceCupformingLeft.R_TRIG_Instance.CLK := FALSE;
   FittingCycle_InstanceCupformingLeft.R_TRIG_Instance.Q := FALSE;
   FittingCycle_InstanceCupformingLeft.R_TRIG_Instance.Stat_Bit := FALSE;
   FittingCycle_InstanceCupformingLeft.H2Reached := TRUE;
   FittingCycle_InstanceCupformingLeft.IEC_Timer_timeout.PT := T#15S;
   FittingCycle_InstanceCupformingLeft.IEC_Timer_timeout.IN := FALSE;
   FittingCycle_InstanceCupformingLeft.DigiforceStarted := TRUE;
   FittingCycle_InstanceCupformingLeft.R_TRIG_Instance_1.CLK := FALSE;
   FittingCycle_InstanceCupformingLeft.R_TRIG_Instance_1.Q := FALSE;
   FittingCycle_InstanceCupformingLeft.R_TRIG_Instance_1.Stat_Bit := FALSE;
   FittingCycle_InstanceCupformingLeft.ton_WayWithTimeoutReached.PT := T#300MS;
   FittingCycle_InstanceCupformingLeft.ton_WayWithTimeoutReached.IN := FALSE;
   FittingCycle_InstanceCupformingRight.parameters.DigiforceProgram := 1;
   FittingCycle_InstanceCupformingRight.parameters.FinalSpeed := 25.0;
   FittingCycle_InstanceCupformingRight.parameters.ApproachSpeed := 25.0;
   FittingCycle_InstanceCupformingRight.parameters.FinalForce := 10.0;
   FittingCycle_InstanceCupformingRight.parameters.ApproachForce := 10.0;
   FittingCycle_InstanceCupformingRight.parameters.EndWayImmediate := 2.7;
   FittingCycle_InstanceCupformingRight.parameters.EndWayWithTimeout := 3.0;
   FittingCycle_InstanceCupformingRight.parameters.SwitchingWay := 20.0;
   FittingCycle_InstanceCupformingRight.parameters.EndWayTimeout := T#300MS;
   FittingCycle_InstanceCupformingRight.basicPosition := TRUE;
   FittingCycle_InstanceCupformingRight.MaxPosition := 105.0;
   FittingCycle_InstanceCupformingRight.endStopCylinderActive := TRUE;
   FittingCycle_InstanceCupformingRight.shiftSupportToWork := TRUE;
   FittingCycle_InstanceCupformingRight.cnt := 0;
   FittingCycle_InstanceCupformingRight.R_TRIG_Instance.CLK := FALSE;
   FittingCycle_InstanceCupformingRight.R_TRIG_Instance.Q := FALSE;
   FittingCycle_InstanceCupformingRight.R_TRIG_Instance.Stat_Bit := FALSE;
   FittingCycle_InstanceCupformingRight.H2Reached := TRUE;
   FittingCycle_InstanceCupformingRight.IEC_Timer_timeout.PT := T#15S;
   FittingCycle_InstanceCupformingRight.IEC_Timer_timeout.IN := FALSE;
   FittingCycle_InstanceCupformingRight.DigiforceStarted := TRUE;
   FittingCycle_InstanceCupformingRight.R_TRIG_Instance_1.CLK := FALSE;
   FittingCycle_InstanceCupformingRight.R_TRIG_Instance_1.Q := FALSE;
   FittingCycle_InstanceCupformingRight.R_TRIG_Instance_1.Stat_Bit := FALSE;
   FittingCycle_InstanceCupformingRight.ton_WayWithTimeoutReached.PT := T#300MS;
   FittingCycle_InstanceCupformingRight.ton_WayWithTimeoutReached.IN := FALSE;
   R_TRIG_Instance.CLK := FALSE;
   R_TRIG_Instance.Q := FALSE;
   R_TRIG_Instance.Stat_Bit := FALSE;
   R_TRIG_Instance_1.CLK := FALSE;
   R_TRIG_Instance_1.Q := FALSE;
   R_TRIG_Instance_1.Stat_Bit := FALSE;
   R_TRIG_Instance_2.CLK := FALSE;
   R_TRIG_Instance_2.Q := FALSE;
   R_TRIG_Instance_2.Stat_Bit := FALSE;
   R_TRIG_Instance_3.CLK := FALSE;
   R_TRIG_Instance_3.Q := FALSE;
   R_TRIG_Instance_3.Stat_Bit := FALSE;
   HydraulicMotor_Instance.cycleActiveCupforming := FALSE;
   HydraulicMotor_Instance.temp1nok := FALSE;
   HydraulicMotor_Instance.temp2nok := FALSE;
   HydraulicMotor_Instance.qKM20 := FALSE;
   HydraulicMotor_Instance.qMotor := FALSE;
   HydraulicMotor_Instance.qValveCupforming := FALSE;
   HydraulicMotor_Instance.R_TRIG_Instance.CLK := FALSE;
   HydraulicMotor_Instance.R_TRIG_Instance.Q := FALSE;
   HydraulicMotor_Instance.R_TRIG_Instance.Stat_Bit := FALSE;
   HydraulicMotor_Instance.cnt := 0;
   HydraulicMotor_Instance.IEC_Timer_0_Instance.PT := T#3S;
   HydraulicMotor_Instance.IEC_Timer_0_Instance.IN := FALSE;
   HydraulicMotor_Instance.F_TRIG_Instance.CLK := FALSE;
   HydraulicMotor_Instance.F_TRIG_Instance.Q := FALSE;
   HydraulicMotor_Instance.F_TRIG_Instance.Stat_Bit := FALSE;
   HydraulicMotor_Instance.IEC_Timer_0_Instance_1.PT := T#0MS;
   HydraulicMotor_Instance.IEC_Timer_0_Instance_1.IN := FALSE;
   dummyCylinderLeft.InWp := FALSE;
   dummyCylinderLeft.InBp := TRUE;
   dummyCylinderLeft.InFp := FALSE;
   dummyCylinderLeft.ToWp := FALSE;
   dummyCylinderLeft.ToBp := TRUE;
   dummyCylinderLeft.ToFp := FALSE;
   dummyCylinderRight.InWp := FALSE;
   dummyCylinderRight.InBp := TRUE;
   dummyCylinderRight.InFp := FALSE;
   dummyCylinderRight.ToWp := FALSE;
   dummyCylinderRight.ToBp := TRUE;
   dummyCylinderRight.ToFp := FALSE;
END_DATA_BLOCK

DATA_BLOCK "ScanCompare_DB"   // DB32
VERSION : 0.1
// stored: AutoNumber true, DBAccessibleFromOPCUA true, DBAccessibleFromWebserver true, InstanceOfName ScanCompare, InstanceOfType FB
"ScanCompare"
   // VAR_INPUT
   //    iDMC : String := '';
   //    iStringToCompare : String := '2567208X';
   //    iPosition : Int := 9;
   //    iLength : Int := 8;
   // END_VAR
   // VAR_OUTPUT
   //    comparedString : String := '';
   //    OK : Bool := FALSE;
   // END_VAR
BEGIN
END_DATA_BLOCK

DATA_BLOCK "RobotJob_DB"   // DB64
VERSION : 0.1
// stored: AutoNumber true, DBAccessibleFromOPCUA true, DBAccessibleFromWebserver true, InstanceOfName RobotJob, InstanceOfType FB
"RobotJob"
BEGIN
END_DATA_BLOCK

DATA_BLOCK "RobotMain_DB"   // DB17
VERSION : 0.1
// stored: AutoNumber true, DBAccessibleFromOPCUA true, DBAccessibleFromWebserver true, InstanceOfName RobotMain, InstanceOfType FB
"RobotMain"
   // VAR_OUTPUT
   //    RobotInStartingPosition : Bool;
   // END_VAR
   // VAR
   //    R1 { S7_SetPoint := 'True'} : "RobotControl";
   //    R_TRIG_Instance { S7_SetPoint := 'True'} : R_TRIG;
   //    F_TRIG_Instance { S7_SetPoint := 'True'} : F_TRIG;
   // END_VAR
BEGIN
   R1.StartReq := FALSE;
   R1.KeyExt := FALSE;
   R1.JobNrReq := 16#00;
   R1.periReady := FALSE;
   R1.stopMess := TRUE;
   R1.progAct := FALSE;
   R1.onPath := FALSE;
   R1.ext := TRUE;
   R1.internalEstop := FALSE;
   R1.home := TRUE;
   R1.pgNoReq := FALSE;
   R1.robStopped := TRUE;
   R1.jobNrBack := 16#00;
   R1.StartAllowed := FALSE;
   R1.Started := FALSE;
   R1.drivesOn := FALSE;
   R1.confMess := FALSE;
   R1.ExtStart := FALSE;
   R1.moveEnable := TRUE;
   R1.reqHome := FALSE;
   R1.pgNoValid := FALSE;
   R1.reqDoor := FALSE;
   R1.jobNr := 16#00;
   R_TRIG_Instance.CLK := FALSE;
   R_TRIG_Instance.Q := FALSE;
   R_TRIG_Instance.Stat_Bit := FALSE;
   F_TRIG_Instance.CLK := FALSE;
   F_TRIG_Instance.Q := FALSE;
   F_TRIG_Instance.Stat_Bit := FALSE;
END_DATA_BLOCK

DATA_BLOCK "Manipulator_main_DB"   // DB42
VERSION : 0.1
// stored: AutoNumber true, DBAccessibleFromOPCUA true, DBAccessibleFromWebserver true, InstanceOfName Manipulator_main, InstanceOfType FB
"Manipulator_main"
BEGIN
END_DATA_BLOCK

DATA_BLOCK "SlidesMain_DB"   // DB45
VERSION : 0.1
// stored: AutoNumber true, DBAccessibleFromOPCUA true, DBAccessibleFromWebserver true, InstanceOfName SlidesMain, InstanceOfType FB
"SlidesMain"
BEGIN
   R_TRIG_Instance.CLK := FALSE;
   R_TRIG_Instance.Q := FALSE;
   R_TRIG_Instance.Stat_Bit := FALSE;
   IEC_Timer_0_Instance.PT := T#0MS;
   IEC_Timer_0_Instance.IN := FALSE;
   IEC_Timer_0_Instance_1.PT := T#0MS;
   IEC_Timer_0_Instance_1.IN := TRUE;
   IEC_Timer_0_Instance_3.PT := T#0MS;
   IEC_Timer_0_Instance_3.IN := FALSE;
   IEC_Timer_0_Instance_5.PT := T#0MS;
   IEC_Timer_0_Instance_5.IN := FALSE;
END_DATA_BLOCK

DATA_BLOCK "ServoMain_DB"   // DB6
VERSION : 0.1
// stored: AutoNumber true, DBAccessibleFromOPCUA true, DBAccessibleFromWebserver true, InstanceOfName ServoMain, InstanceOfType FB
"ServoMain"
BEGIN
END_DATA_BLOCK

DATA_BLOCK "DB_INST_AWAKE_SIGNAL"   // DB1003
VERSION : 0.1
// stored: AutoNumber false, DBAccessibleFromOPCUA true, DBAccessibleFromWebserver true, InstanceOfName FB_IJC_AWAKE_SIGNAL, InstanceOfType FB
"FB_IJC_AWAKE_SIGNAL"
BEGIN
END_DATA_BLOCK

DATA_BLOCK "7. Call_M103_PY_DB"   // DB82
VERSION : 0.1
// stored: AutoNumber true, DBAccessibleFromOPCUA true, DBAccessibleFromWebserver true, InstanceOfName 7. Call_M103_PY, InstanceOfType FB
"7. Call_M103_PY"
BEGIN
END_DATA_BLOCK

DATA_BLOCK "IEC_Timer_0_DB_1"   // DB78
{ S7_Optimized_Access := 'TRUE' }
// stored: AutoNumber true, DBAccessibleFromOPCUA true, DBAccessibleFromWebserver true, InstanceOfName IEC_TIMER, OfSystemLibElement IEC_TIMER, OfSystemLibVersion 1.0
"IEC_TIMER"
   // VAR
   //    PT : Time;
   //    ET { ExternalWritable := 'False'} : Time;
   //    IN : Bool;
   //    Q { ExternalWritable := 'False'} : Bool;
   // END_VAR
BEGIN
END_DATA_BLOCK

DATA_BLOCK "SET_TIMEZONE_DB"   // DB5
// stored: AutoNumber true, DBAccessibleFromOPCUA true, DBAccessibleFromWebserver true, InstanceOfName SET_TIMEZONE, OfSystemLibElement SET_TIMEZONE, OfSystemLibVersion 2.0
"SET_TIMEZONE"
   // VAR_INPUT
   //    REQ { ExternalAccessible := 'False'; ExternalVisible := 'False'; ExternalWritable := 'False'} : Bool;
   //    TimeZone { ExternalAccessible := 'False'; ExternalVisible := 'False'; ExternalWritable := 'False'} : TimeTransformationRule;
   // END_VAR
   // VAR_OUTPUT
   //    DONE : Bool;
   //    BUSY : Bool;
   //    ERROR : Bool;
   //    STATUS : Word;
   // END_VAR
   // VAR
   //    BusyState : Word;
   //    LastScanREQ { S7_SetPoint := 'True'} : Bool;
   // END_VAR
BEGIN
END_DATA_BLOCK

DATA_BLOCK "READER_FRONT_TUBE"   // DB72
VERSION : 0.1
// stored: AutoNumber true, DBAccessibleFromOPCUA true, DBAccessibleFromWebserver true, InstanceOfName READER_LOGIC, InstanceOfType FB
"READER_LOGIC"
BEGIN
END_DATA_BLOCK

DATA_BLOCK "READER_REAR_TUBE"   // DB76
VERSION : 0.1
// stored: AutoNumber true, DBAccessibleFromOPCUA true, DBAccessibleFromWebserver true, InstanceOfName READER_LOGIC, InstanceOfType FB
"READER_LOGIC"
BEGIN
END_DATA_BLOCK

DATA_BLOCK "READER_SIDE_LH"   // DB71
VERSION : 0.1
// stored: AutoNumber true, DBAccessibleFromOPCUA true, DBAccessibleFromWebserver true, InstanceOfName READER_LOGIC, InstanceOfType FB
"READER_LOGIC"
BEGIN
END_DATA_BLOCK

DATA_BLOCK "READER_SIDE_RH"   // DB70
VERSION : 0.1
// stored: AutoNumber true, DBAccessibleFromOPCUA true, DBAccessibleFromWebserver true, InstanceOfName READER_LOGIC, InstanceOfType FB
"READER_LOGIC"
BEGIN
END_DATA_BLOCK

DATA_BLOCK "DB_INST_READINGS"   // DB300
VERSION : 0.1
// stored: AutoNumber false, DBAccessibleFromOPCUA true, DBAccessibleFromWebserver true, InstanceOfName FB_READINGS, InstanceOfType FB
"FB_READINGS"
BEGIN
END_DATA_BLOCK

DATA_BLOCK "0. OpcUaClient_DB"   // DB2000
AUTHOR : SiemensAG
VERSION : 1.0
// stored: AutoNumber false, DBAccessibleFromOPCUA true, DBAccessibleFromWebserver true, InstanceOfName 0. OpcUaClient, InstanceOfType FB
"0. OpcUaClient"
BEGIN
END_DATA_BLOCK

DATA_BLOCK "1. DMC_setConnection_DB"   // DB2002
VERSION : 0.1
// stored: AutoNumber false, DBAccessibleFromOPCUA true, DBAccessibleFromWebserver true, InstanceOfName 1. DMC_setConnection, InstanceOfType FB
"1. DMC_setConnection"
BEGIN
END_DATA_BLOCK

DATA_BLOCK "2. Call_M000_PRODUCTION_DECLARATION_DB"   // DB2003
VERSION : 0.1
// stored: AutoNumber false, DBAccessibleFromOPCUA true, DBAccessibleFromWebserver true, InstanceOfName 2. Call_M000_PRODUCTION_DECLARATION, InstanceOfType FB
"2. Call_M000_PRODUCTION_DECLARATION"
BEGIN
END_DATA_BLOCK

DATA_BLOCK "2. Call_M000_PRODUCTION_DECLARATION_DB_1"   // DB2004
VERSION : 0.1
// stored: AutoNumber false, DBAccessibleFromOPCUA true, DBAccessibleFromWebserver true, InstanceOfName 2. Call_M000_PRODUCTION_DECLARATION, InstanceOfType FB
"2. Call_M000_PRODUCTION_DECLARATION"
BEGIN
END_DATA_BLOCK

DATA_BLOCK "5. Call_M005_VARIABILITY_DB"   // DB2005
VERSION : 0.1
// stored: AutoNumber false, DBAccessibleFromOPCUA true, DBAccessibleFromWebserver true, InstanceOfName 5. Call_M005_VARIABILITY, InstanceOfType FB
"5. Call_M005_VARIABILITY"
BEGIN
END_DATA_BLOCK

DATA_BLOCK "6. Call_M004_NTRS_DB"   // DB81
VERSION : 0.1
// stored: AutoNumber true, DBAccessibleFromOPCUA true, DBAccessibleFromWebserver true, InstanceOfName 6. Call_M004_NTRS, InstanceOfType FB
"6. Call_M004_NTRS"
BEGIN
END_DATA_BLOCK

DATA_BLOCK "DB_INST_DTM_READERS"   // DB77
VERSION : 0.1
// stored: AutoNumber true, DBAccessibleFromOPCUA true, DBAccessibleFromWebserver true, InstanceOfName FB_DTM_READERS, InstanceOfType FB
"FB_DTM_READERS"
BEGIN
END_DATA_BLOCK
